INTERFACE I_NAME

PROPERTY Name : STRING
GET
END_GET
SET
END_SET
END_PROPERTY

METHOD NUM : INT
VAR_INPUT
END_VAR
END_METHOD

END_INTERFACE

(* stored: Version 1.1.0.1, ProductVersion 3.1.4024.3
   Itf I_NAME: Id {bb4b401a-6956-4680-8b69-f4664edb99b3}
   Property Name: Id {74e0c294-fead-4aa2-a47c-0ea6d351dbff}
   Get Get: Id {04b5ef29-d27e-4063-85ab-0a09d0f2bf13}
   Set Set: Id {ad5cfa94-0a58-45d3-b3af-c6394b5fe8cf}
   Method NUM: Id {5d388964-ccde-4860-b785-be73ee478113} *)
